{attribute 'qualified_only'}
VAR_GLOBAL
	
	

	// Actual Temperature
	fTempActual: REAL := 0.5;
	// Set Temperature
	fTempSet: REAL := 0.2;
	// Door Status
	bDoorOpen: BOOL := FALSE;
	// Compressor Running Time After Which an Alarm Sounds
	tlmAlarmThreshold: TIME := T#30s;
	// Time from door opening after which alarm sounds
	tDoorOPenThreshold: TIME := T#10s;
	// Control Signal
	xCompressor: BOOL := FALSE;
	// Control Signal
	xSignal: BOOL := FALSE;
	// Status Message
	xLamp: BOOL := FALSE;
	// Ouput for controlling the compressor
	bCompressor: BOOL := FALSE;
	// Output for controlling signal
	bSingal: BOOL := FALSE;
	// Output for controlling the lamp
	bLamp: BOOL := FALSE;
END_VAR

(* stored: Version 1.1.0.1, ProductVersion 3.1.4024.12
   GVL GVL_VAR: Id {bfa1e441-34ab-431e-bd1c-bba2646486f7} *)
